FUNCTION_BLOCK FB_HighVoltage
VAR_INPUT
	i_xExtIlkOK	:	BOOL; //External Interlock, SET to TRUE if not used
END_VAR
VAR_OUTPUT
	{attribute 'pytmc' := '
    pv:
	'}
	hv:ST_HV;
END_VAR
VAR
	(*outputs*)
	q_HV_DO AT %Q*: BOOL;
END_VAR


hv.xIlkOK := i_xExtIlkOK;

q_HV_DO := hv.HV_sw AND hv.xIlkOK;

(*soft io mapping*)
hv.q_HV_DO := q_HV_DO;

END_FUNCTION_BLOCK

(* stored: Version 1.1.0.1, ProductVersion 3.1.4022.12
   POU FB_HighVoltage: Id {18f48132-2f8b-4bad-b9a5-e87aec49b8a9}, SpecialFunc None *)
